PROGRAM MAIN
VAR_INPUT
END_VAR
VAR
	ExecuteSection1 : FB_EXECUTE_SECTION1;
	ExecuteSection2 : FB_EXECUTE_SECTION2;
	ActiveTestStage : INT := 0;
	tDelay : TON;
    bDelayDone : BOOL;
END_VAR



CASE ActiveTestStage OF
	
	0: // Idle
		GVL.GO_HOME := TRUE;
		IF GVL.HMI_BEGIN_TEST THEN
			// user pressed "BEGIN Test"
			ActiveTestStage := 1;
			GVL.HMI_BEGIN_TEST := FALSE;
		END_IF
	
		
		
	1: 
		// Run Section1
		WRITE_IO_VALUES();
		ExecuteSection1(StartTest := TRUE);
		
		// Log Section1
		IF ExecuteSection1.Done THEN
			GVL.HMI_SECTION_1_COMPLETE := TRUE;
			LOG_SECTION1();
			ActiveTestStage := 2;
		END_IF
		
	2: 
		GVL.HMI_SECTION_2_INSTRUCTIONS := 'Open JBOX DOOR, PRESS ESTOP, PULL FIRE ALARM HANDLE';
		IF GVL.HMI_BEGIN_SECTION_2 THEN
			HMI_BEGIN_SECTION_2 := FALSE;
			WRITE_IO_VALUES();
			ExecuteSection2(StartTest := TRUE);
			IF ExecuteSection2.Done THEN
				GVL.HMI_SECTION_2_COMPLETE := TRUE;
				LOG_SECTION2();
				ActiveTestStage := 999;
			END_IF
		END_IF
		
	999: // Test done
		GVL.TESTING_PROGRAM_COMPLETE := TRUE;

		
		
END_CASE

IF GVL.HMI_RESET_TEST THEN
    GVL.ABORT_SUCCESSFUL := UNINITIALIZE();
	tDelay(IN := TRUE, PT := T#3S);
	
	bDelayDone := tDelay.Q;
	IF bDelayDone THEN
		GVL.ABORT_SUCCESSFUL := FALSE;
    	GVL.HMI_RESET_TEST := FALSE;
		ActiveTestStage := 0;
	END_IF;
	

END_IF

END_PROGRAM

(* stored: Version 1.1.0.1, ProductVersion 3.1.4024.10
   POU MAIN: Id {99ab54a4-34ac-447e-8e15-602a1f030758}, SpecialFunc None *)
